{attribute 'qualified_only'}
VAR_GLOBAL
END_VAR

(* stored: Version 1.1.0.1
   GVL Safety: Id {6a582cab-e4d6-423c-b57e-300a55c0abfe} *)
